{attribute 'GeneratedUsingTerminal: AT2020-0250-0019'}
{attribute addProperty BoxType "AT2020-0250-0019"}
{attribute addProperty Id "ControlAT %Q*UINT2Current_setpoint_value_ChAT %Q*ARRAY[0..14] OF INT30"}
{attribute addProperty CRC "3100183749"}
{attribute addProperty Size "32"}
TYPE CC_Outputs_69F9BE14 :
STRUCT
	{attribute addProperty Name "Control"}
	Control AT %Q* : UINT;
	{attribute addProperty Name "Current_setpoint_value_Ch"}
	Current_setpoint_value_Ch AT %Q* : ARRAY[0..14] OF INT;
END_STRUCT
END_TYPE

(* stored: Version 1.2.0.0, ProductVersion 3.1.4024.9
   DUT CC_Outputs_69F9BE14: Id {78df9af2-840d-43f9-a87b-752e95838fbf} *)
